FUNCTION_BLOCK FB_011WriteRParameter

VAR_INPUT
	Execute:BOOL;
	fbnChannelid:UDINT;
	nRParamAry:ARRAY[0..19] OF LREAL;
END_VAR
VAR_OUTPUT
END_VAR
VAR
	fbWriteRParams:ItpWriteRParams;
END_VAR


fbWriteRParams(
	bExecute:= Execute, 
	nChnId:= fbnChannelid, 
	pAddr:= ADR(nRParamAry), 
	nIndex:= 0, 
	nCount:= 10, 
	tTimeOut:= T#2S, 
	bBusy=> , 
	bErr=> , 
	nErrId=> );

END_FUNCTION_BLOCK

(* stored: Version 1.1.0.1, ProductVersion 3.1.4024.12
   POU FB_011WriteRParameter: Id {96ae41d8-aad3-443f-b1ad-b24402477985}, SpecialFunc None *)
